FUNCTION_BLOCK FB_PipelineConsumer
VAR
    stage : B4Pipeline_Plc.FB_PipelineStage;
    bStageError : BOOL;
END_VAR

stage(value := -1);
bStageError := stage.bError;

END_FUNCTION_BLOCK

(* stored: Version 1.1.0.1
   POU FB_PipelineConsumer: Id {bf5f8c6f-78c6-457d-978d-4572836a1b84}, SpecialFunc None *)
